// TIA Portal V18 export
// export: Created 2026-06-08T16:32:20.6921849Z, ExportSetting WithDefaults, DisplayName Totally Integrated Automation Portal, DisplayVersion V18, DisplayName TIA Portal Openness, DisplayVersion V18, DisplayName TIA Portal Version Control Interface, DisplayVersion V18, DisplayName STEP 7 Professional, DisplayVersion V18, DisplayName STEP 7 Safety, DisplayVersion V18, DisplayName WinCC Professional, DisplayVersion V18
FUNCTION_BLOCK "LID_execess_remove_station"   // FB4, LAD
VERSION : 0.1
// stored: AutoNumber true, IsIECCheckEnabled false, UDAEnableTagReadback false
   VAR_TEMP   // added for the SCL form of the ladder/FBD networks
      _w1 : Bool;
   END_VAR
BEGIN

REGION Network 1: LID_BELT_EXECESS_CONVYR_HANDLER
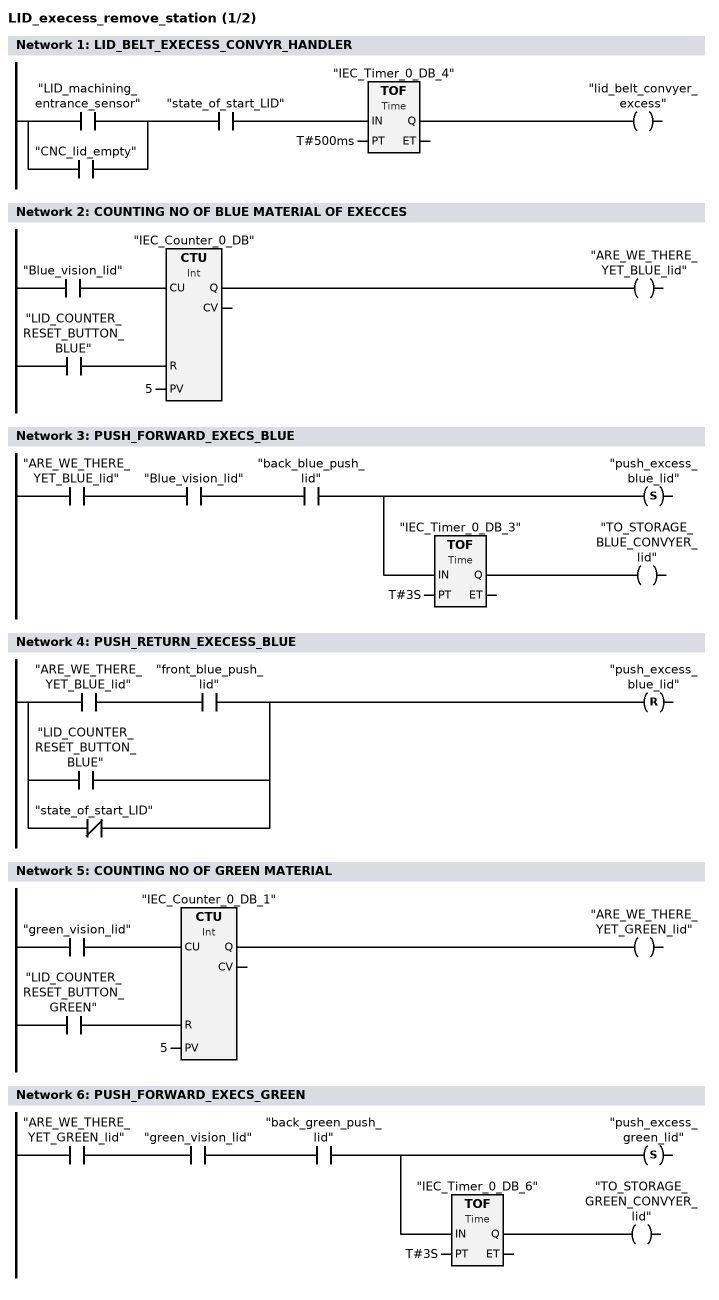
   RUNG wire#powerrail
      Contact( "LID_machining_entrance_sensor" )
      wire#w1
      Contact( "state_of_start_LID" )
      { S7_Templates := "time_type := Time" } "IEC_Timer_0_DB_4".TOF(pt := T#500ms, et =>)
      Coil( "lid_belt_convyer_excess" )
   END_RUNG
   RUNG wire#powerrail
      Contact( "CNC_lid_empty" )
   END_RUNG wire#w1
   // the same network as SCL:
   "IEC_Timer_0_DB_4".TOF(IN := ("LID_machining_entrance_sensor" OR "CNC_lid_empty") AND "state_of_start_LID",
                          PT := T#500ms);
   "lid_belt_convyer_excess" := "IEC_Timer_0_DB_4".Q;
END_REGION

REGION Network 2: COUNTING NO OF BLUE MATERIAL OF EXECCES
   RUNG wire#powerrail
      Contact( "Blue_vision_lid" )
      { S7_Templates := "value_type := Int" } "IEC_Counter_0_DB".CTU(r := wire#w1, pv := 5, cv =>)
      Coil( "ARE_WE_THERE_YET_BLUE_lid" )
   END_RUNG
   RUNG wire#powerrail
      Contact( "LID_COUNTER_RESET_BUTTON_BLUE" )
   END_RUNG wire#w1
   // the same network as SCL:
   "IEC_Counter_0_DB".CTU(CU := "Blue_vision_lid", R := "LID_COUNTER_RESET_BUTTON_BLUE", PV := 5);
   "ARE_WE_THERE_YET_BLUE_lid" := "IEC_Counter_0_DB".Q;
END_REGION

REGION Network 3: PUSH_FORWARD_EXECS_BLUE
   RUNG wire#powerrail
      Contact( "ARE_WE_THERE_YET_BLUE_lid" )
      Contact( "Blue_vision_lid" )
      Contact( "back_blue_push_lid" )
      wire#w1
      S_Coil( "push_excess_blue_lid" )
   END_RUNG
   RUNG wire#w1
      { S7_Templates := "time_type := Time" } "IEC_Timer_0_DB_3".TOF(pt := T#3S, et =>)
      Coil( "TO_STORAGE_BLUE_CONVYER_lid" )
   END_RUNG
   // the same network as SCL:
   #_w1 := "ARE_WE_THERE_YET_BLUE_lid" AND "Blue_vision_lid" AND "back_blue_push_lid";
   IF #_w1 THEN "push_excess_blue_lid" := TRUE; END_IF;
   "IEC_Timer_0_DB_3".TOF(IN := #_w1, PT := T#3S);
   "TO_STORAGE_BLUE_CONVYER_lid" := "IEC_Timer_0_DB_3".Q;
END_REGION

REGION Network 4: PUSH_RETURN_EXECESS_BLUE
   RUNG wire#powerrail
      Contact( "ARE_WE_THERE_YET_BLUE_lid" )
      Contact( "front_blue_push_lid" )
      wire#w1
      R_Coil( "push_excess_blue_lid" )
   END_RUNG
   RUNG wire#powerrail
      Contact( "LID_COUNTER_RESET_BUTTON_BLUE" )
   END_RUNG wire#w1
   RUNG wire#powerrail
      I_Contact( "state_of_start_LID" )
   END_RUNG wire#w1
   // the same network as SCL:
   IF ("ARE_WE_THERE_YET_BLUE_lid" AND "front_blue_push_lid") OR "LID_COUNTER_RESET_BUTTON_BLUE" OR NOT "state_of_start_LID" THEN
       "push_excess_blue_lid" := FALSE;
   END_IF;
END_REGION

REGION Network 5: COUNTING NO OF GREEN MATERIAL
   RUNG wire#powerrail
      Contact( "green_vision_lid" )
      { S7_Templates := "value_type := Int" } "IEC_Counter_0_DB_1".CTU(r := wire#w1, pv := 5, cv =>)
      Coil( "ARE_WE_THERE_YET_GREEN_lid" )
   END_RUNG
   RUNG wire#powerrail
      Contact( "LID_COUNTER_RESET_BUTTON_GREEN" )
   END_RUNG wire#w1
   // the same network as SCL:
   "IEC_Counter_0_DB_1".CTU(CU := "green_vision_lid", R := "LID_COUNTER_RESET_BUTTON_GREEN", PV := 5);
   "ARE_WE_THERE_YET_GREEN_lid" := "IEC_Counter_0_DB_1".Q;
END_REGION

REGION Network 6: PUSH_FORWARD_EXECS_GREEN
   RUNG wire#powerrail
      Contact( "ARE_WE_THERE_YET_GREEN_lid" )
      Contact( "green_vision_lid" )
      Contact( "back_green_push_lid" )
      wire#w1
      S_Coil( "push_excess_green_lid" )
   END_RUNG
   RUNG wire#w1
      { S7_Templates := "time_type := Time" } "IEC_Timer_0_DB_6".TOF(pt := T#3S, et =>)
      Coil( "TO_STORAGE_GREEN_CONVYER_lid" )
   END_RUNG
   // the same network as SCL:
   #_w1 := "ARE_WE_THERE_YET_GREEN_lid" AND "green_vision_lid" AND "back_green_push_lid";
   IF #_w1 THEN "push_excess_green_lid" := TRUE; END_IF;
   "IEC_Timer_0_DB_6".TOF(IN := #_w1, PT := T#3S);
   "TO_STORAGE_GREEN_CONVYER_lid" := "IEC_Timer_0_DB_6".Q;
END_REGION

REGION Network 7: PUSH_RETURN_GREEN
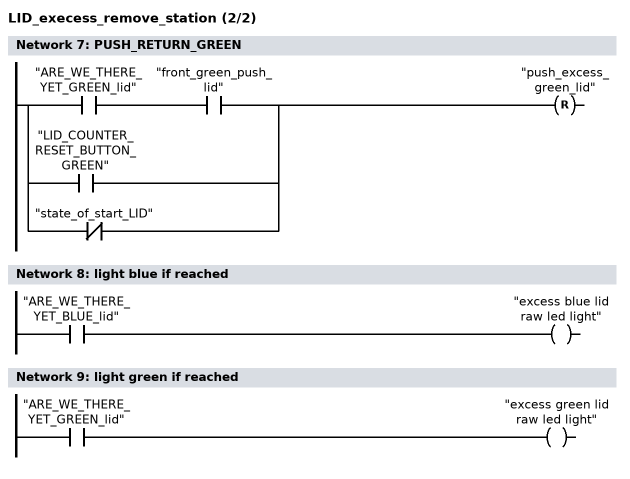
   RUNG wire#powerrail
      Contact( "ARE_WE_THERE_YET_GREEN_lid" )
      Contact( "front_green_push_lid" )
      wire#w1
      R_Coil( "push_excess_green_lid" )
   END_RUNG
   RUNG wire#powerrail
      Contact( "LID_COUNTER_RESET_BUTTON_GREEN" )
   END_RUNG wire#w1
   RUNG wire#powerrail
      I_Contact( "state_of_start_LID" )
   END_RUNG wire#w1
   // the same network as SCL:
   IF ("ARE_WE_THERE_YET_GREEN_lid" AND "front_green_push_lid") OR "LID_COUNTER_RESET_BUTTON_GREEN" OR NOT "state_of_start_LID" THEN
       "push_excess_green_lid" := FALSE;
   END_IF;
END_REGION

REGION Network 8: light blue if reached
   RUNG wire#powerrail
      Contact( "ARE_WE_THERE_YET_BLUE_lid" )
      Coil( "excess blue lid raw led light" )
   END_RUNG
   // the same network as SCL:
   "excess blue lid raw led light" := "ARE_WE_THERE_YET_BLUE_lid";
END_REGION

REGION Network 9: light green if reached
   RUNG wire#powerrail
      Contact( "ARE_WE_THERE_YET_GREEN_lid" )
      Coil( "excess green lid raw led light" )
   END_RUNG
   // the same network as SCL:
   "excess green lid raw led light" := "ARE_WE_THERE_YET_GREEN_lid";
END_REGION
END_FUNCTION_BLOCK
